Yaskawa INFORM job: BATMAN-40.JBI

/JOB
//NAME BATMAN-40
///FOLDERNAME OBROTNIK
//POS
///NPOS 0,0,1,0,0,0
///TOOL 0
///POSTYPE PULSE
///PULSE
EC00000=-363194,-550745
//INST
///DATE 2023/12/20 10:03
///ATTR SC,RW,RJ
////FRAME ROBOT
///GROUP1 ST1
NOP
MOVJ EC00000 VJ=100.00
END
